INTERFACE I_HwTimestamp_Mode EXTENDS __SYSTEM.IQueryInterface

{attribute 'monitoring' := 'call'}
PROPERTY Duration_1us : UDINT
GET
END_GET
SET
END_SET
END_PROPERTY

METHOD PUBLIC Trigger : HRESULT
VAR_INPUT
	//The data type T_DCTIME64 represents the distributed clock system time (abbreviated as DC time) as a linear 64-bit integer value. 
	//The time is expressed in nanoseconds since 1/1/2000 UTC. The smallest unit is a nanosecond.
	//F_GetCurDcTickTime64()
	nDCTimeStamp	: T_DCTIME64;
END_VAR
END_METHOD

{attribute 'monitoring' := 'call'}
// The given trigger time is delayed by this value. E.g. to wait for the maximum lighting value before taking a picture  [in 1ns]
PROPERTY TriggerDelay_1ns : UDINT
GET
END_GET
SET
END_SET
END_PROPERTY

END_INTERFACE

(* stored: Version 1.1.0.1, ProductVersion 3.1.4024.12
   Itf I_HwTimestamp_Mode: Id {94b0a5e6-77b2-4f2e-b5e0-efb47bca32c9}
   Property Duration_1us: Id {5f15678e-69c1-42b4-b23c-be8c8395eefd}
   Get Get: Id {3d7b3b9b-14b1-4625-a95f-241cc21c013e}
   Set Set: Id {b2d1ebae-882f-4849-8a91-5b96e0219679}
   Method Trigger: Id {a6220490-d492-41e0-904d-1812b526ed46}
   Property TriggerDelay_1ns: Id {2a522584-211a-4538-b0eb-5cdc7a741441}
   Get Get: Id {8575f761-4e07-4e9e-a343-c1e71b5ad62d}
   Set Set: Id {7cff1531-0450-4255-91c5-c98514566c9d} *)
